FUNCTION_BLOCK Conveyor_4 (* Basic Function Block Type *)
  (* Standard: 61499-2 *)
  (* Version 0.2, 2003-12-04, JHC, Rockwell Automation, Renamed for better indexing. *)
  (* Version 0.1, 2002-11-05, JHC, Rockwell Automation, Corrected missing ST element in Algorithm REQ. *)
  (* Version 0.0, 2000-05-30, JHC, Rockwell Automation *)
  (* Compiler header: package fb.rt.cs725; *)
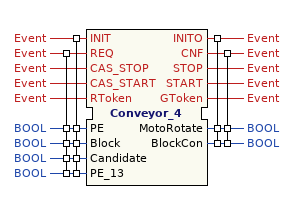
  EVENT_INPUT
    INIT WITH PE, Block, Candidate, PE_13; (* Initialization Request *)
    REQ WITH PE, Block, Candidate, PE_13; (* Normal Execution Request *)
    CAS_STOP;
    CAS_START;
    RToken;
  END_EVENT
  EVENT_OUTPUT
    INITO WITH MotoRotate, BlockCon; (* Initialization Confirm *)
    CNF WITH MotoRotate, BlockCon; (* Execution Confirmation *)
    STOP;
    START;
    GToken;
  END_EVENT
  VAR_INPUT
    PE : BOOL; (* Input event qualifier *)
    Block : BOOL;
    Candidate : BOOL;
    PE_13 : BOOL;
  END_VAR
  VAR_OUTPUT
    MotoRotate : BOOL; (* Output event qualifier *)
    BlockCon : BOOL;
  END_VAR
  VAR
    lastPE : BOOL := 1;
    lastBlock : BOOL := 0;
  END_VAR
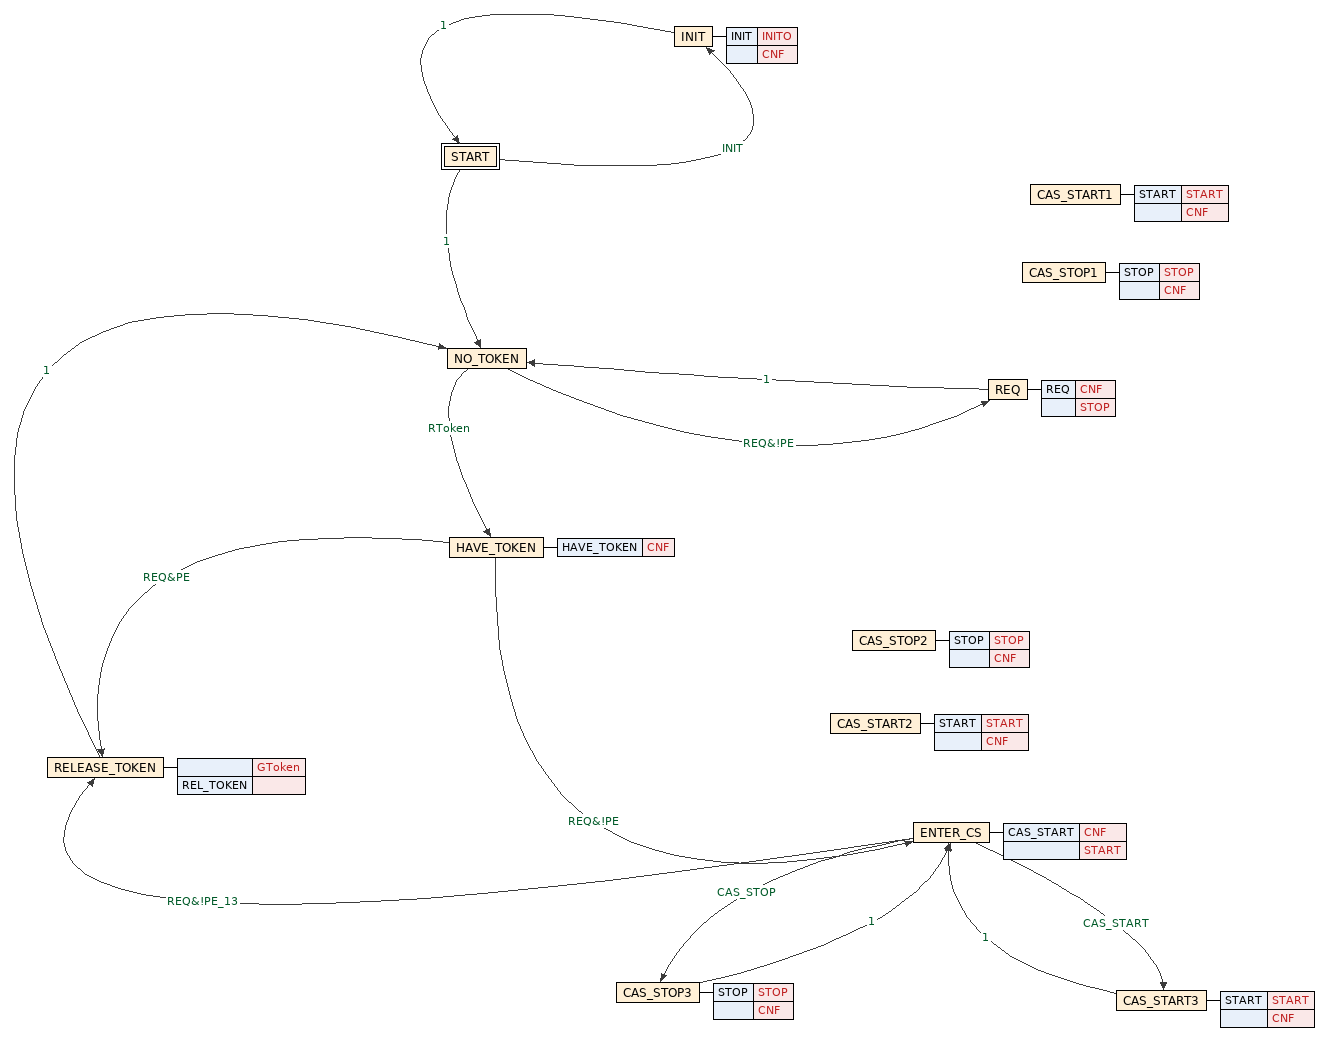
  EC_STATES
    START; (* Initial State *)
    INIT : INIT -> INITO, -> CNF; (* Initialization *)
    REQ : REQ -> CNF, -> STOP; (* Normal execution *)
    ENTER_CS : CAS_START -> CNF, -> START;
    RELEASE_TOKEN : -> GToken, REL_TOKEN;
    NO_TOKEN;
    HAVE_TOKEN : HAVE_TOKEN -> CNF;
    CAS_START1 : START -> START, -> CNF;
    CAS_STOP1 : STOP -> STOP, -> CNF;
    CAS_START2 : START -> START, -> CNF;
    CAS_STOP2 : STOP -> STOP, -> CNF;
    CAS_START3 : START -> START, -> CNF;
    CAS_STOP3 : STOP -> STOP, -> CNF;
  END_STATES
  EC_TRANSITIONS
    START TO INIT := INIT;
    INIT TO START := 1;
    START TO NO_TOKEN := 1;
    NO_TOKEN TO HAVE_TOKEN := RToken;
    HAVE_TOKEN TO RELEASE_TOKEN := REQ&PE;
    NO_TOKEN TO REQ := REQ&!PE;
    REQ TO NO_TOKEN := 1;
    HAVE_TOKEN TO ENTER_CS := REQ&!PE;
    RELEASE_TOKEN TO NO_TOKEN := 1;
    ENTER_CS TO RELEASE_TOKEN := REQ&!PE_13;
    ENTER_CS TO CAS_START3 := CAS_START;
    CAS_START3 TO ENTER_CS := 1;
    CAS_STOP3 TO ENTER_CS := 1;
    ENTER_CS TO CAS_STOP3 := CAS_STOP;
  END_TRANSITIONS
  ALGORITHM INIT IN Java: (* Initialization algorithm *)
MotoRotate.value=true;
Block.value=false;

System.out.println(this+" "+MotoRotate.value);
System.out.println(MotoRotate.value);
  END_ALGORITHM
  ALGORITHM REQ IN Java: (* Normally executed algorithm *)
System.out.println("BAG DETECTED!!");
MotoRotate.value=false;
  END_ALGORITHM
  ALGORITHM START IN Java:
MotoRotate.value=true;
  END_ALGORITHM
  ALGORITHM STOP IN Java:
MotoRotate.value=false;
  END_ALGORITHM
  ALGORITHM CAS_START IN Java:
System.out.println("Starting again");
System.out.println("Token received");
MotoRotate.value=true;
  END_ALGORITHM
  ALGORITHM REL_TOKEN IN Java:
System.out.println("Released token from c4");
  END_ALGORITHM
  ALGORITHM HAVE_TOKEN IN Java:
System.out.println("Have the token");
  END_ALGORITHM
END_FUNCTION_BLOCK
